Yaskawa INFORM job: BALON_1.JBI

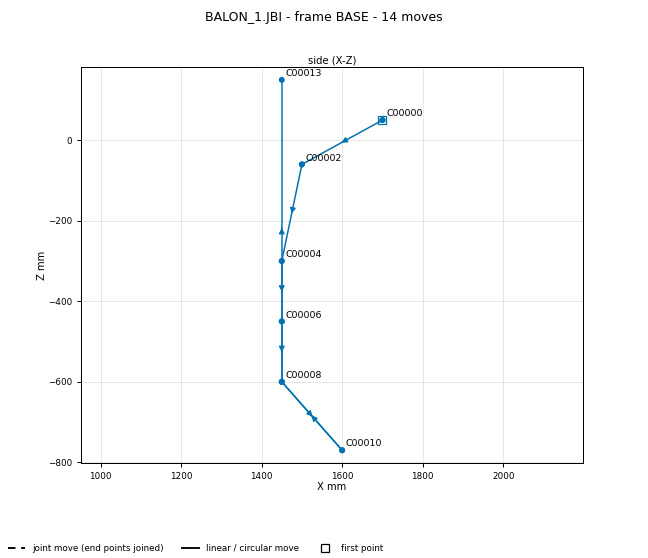
[picture p0: tool path of BALON_1.JBI in frame BASE, 14 of 14 moves have a stored position in this frame; points joined in program order, loops and branches not executed]
/JOB
//NAME BALON_1
//POS
///NPOS 14,0,14,0,0,0
///TOOL 0
///POSTYPE BASE
///RECTAN
///RCONF 0,0,0,0,0,0,0,0,0,0,0,0,0,0,0,0,0,0,0,0,0,0,0,0
C00000=1700.000,35.000,50.000,-180.0000,-30.0000,0.0000
C00001=1700.000,35.000,50.000,-180.0000,-30.0000,0.0000
C00002=1500.000,35.000,-60.000,180.0000,-50.0000,0.0000
C00003=1500.000,35.000,-60.000,180.0000,-50.0000,0.0000
C00004=1450.000,35.000,-300.000,-100.0000,-90.0000,-75.0000
C00005=1450.000,35.000,-300.000,-100.0000,-90.0000,-75.0000
C00006=1450.000,35.000,-450.000,-100.0000,-90.0000,-75.0000
C00007=1450.000,35.000,-450.000,-100.0000,-90.0000,-75.0000
C00008=1450.000,35.000,-600.000,-100.0000,-90.0000,-75.0000
C00009=1450.000,35.000,-600.000,-100.0000,-90.0000,-75.0000
C00010=1600.000,35.000,-770.000,-180.0000,-75.0000,0.0000
C00011=1600.000,35.000,-770.000,-180.0000,-75.0000,0.0000
C00012=1450.000,35.000,-600.000,-100.0000,-90.0000,-75.0000
C00013=1450.000,35.000,150.000,-100.0000,-90.0000,-75.0000
///POSTYPE PULSE
///PULSE
EC00000=0
EC00001=370000
EC00002=370000
EC00003=0
EC00004=0
EC00005=370000
EC00006=370000
EC00007=0
EC00008=0
EC00009=370000
EC00010=370000
EC00011=0
EC00012=0
EC00013=0
//INST
///DATE 2023/04/18 16:39
///ATTR SC,RW,RJ
////FRAME BASE
///GROUP1 RB1,ST1
NOP
MOVJ C00000 EC00000 VJ=15.00
CALL JOB:SPYON
MOVJ C00001 EC00001 VJ=12.00
MOVL C00002 EC00002 V=200.0
MOVJ C00003 EC00003 VJ=12.00
MOVL C00004 EC00004 V=200.0
MOVJ C00005 EC00005 VJ=12.00
MOVL C00006 EC00006 V=200.0
MOVJ C00007 EC00007 VJ=12.00
MOVL C00008 EC00008 V=200.0
MOVJ C00009 EC00009 VJ=12.00
MOVL C00010 EC00010 V=200.0
MOVJ C00011 EC00011 VJ=12.00
CALL JOB:SPYOF
MOVL C00012 EC00012 V=150.0
MOVL C00013 EC00013 V=150.0
END
